# B&R Automation Studio project KeePakST401VersionX
Automation Studio 4.7.5.60 SP; technology packages: Acp10Arnc0 5.8.2, mapp 1.71.0, TextSystem 

## Configuration Config1

CPU X20CP0484, AutomationRuntime C4.72, Build 4.1.2, Vc V4.72.0

### Task classes (Cpu.sw)
```
Cyclic#4 (cycle 100000 us, tolerance 100000 us):
  Program <- Program.prg
  FlexTest <- Actuators.FlexTest.prg
Libraries: AsEPL, runtime, AsBrStr, AsMbTCP, standard, Lib_PBFlx
```

### Hardware
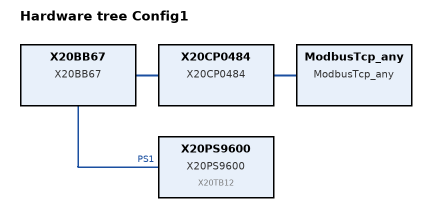
```
ModbusTcp_any : ModbusTcp_any v1.0.6.0  [ETH1 -> X20CP0484.IF2 [Cable Type=PowerlinkCable, Length=10, Version=1.0.0.2]]
  IpAddress = 192.168.0.56
  UnitId = 1
X20BB67 : X20BB67 v1.1.0.0
  Connector IF6:
    CycleTime = 4000
X20CP0484 : X20CP0484 v1.2.1.0  [SL -> X20BB67.SL1]
  Connector IF2:
    ActivateDevice = 1
    Mode = Manual
    InternetAddress = 192.168.0.137
    SubnetMask = 255.255.255.0
    InaNodeNumber = 3
    ActivateModbus = 1
    NumSlaves = -1
    NumAllBlocks = -1
    MemSizeIn = -1
    MemSizeOut = -1
    SlaveDiagnostics = 1
  ConfigurationID = PBFlex_PL_Test1_Config1
  TimerDeviceType = SWIOTIMER
  Cyclic1Duration = 10000
  Cyclic1Tolerance = 10000
  Cyclic2Duration = 20000
  Cyclic2Tolerance = 20000
  Cyclic3Duration = 50000
  Cyclic3Tolerance = 50000
  Cyclic4Duration = 100000
  Cyclic4Tolerance = 100000
  Cyclic5Duration = 200000
  Cyclic5Tolerance = 200000
  Cyclic6Duration = 500000
  Cyclic6Tolerance = 500000
  Cyclic7Duration = 1000000
  Cyclic7Tolerance = 1000000
  Cyclic8Duration = 10000
  Cyclic8Tolerance = 30000000
X20PS9600 : X20PS9600 v1.0.1.0  [PS -> X20BB67.PS1; SS1 -> X20TB12.SS]
X20TB12 : X20TB12 v1.0.0.0
```

### IoMap.iom - X20CP0484/IoMap.iom
```iecst
VAR_CONFIG
	::i_arr_Input_Flex[0] AT %IW."ModbusTcp_any".StateData1;
	::i_arr_Input_Flex[1] AT %IW."ModbusTcp_any".StateData2;
	::i_arr_Output_Flex[0] AT %QW."ModbusTcp_any".CtrWord;
	::b_ModuleStatus AT %IX."ModbusTcp_any".ModuleOk;
END_VAR
```

## Configuration MasterConfiguration_ServoRam

CPU X20CP0484, AutomationRuntime C4.72, Build 4.1.2, Safety 1.10, Vc V4.72.0

### Task classes (Cpu.sw)
```
Cyclic#1 (cycle 4000 us, tolerance 0 us):
  ModeContro <- ModeControl.ModeControl_ST.prg
Cyclic#2 (cycle 8000 us, tolerance 8000 us):
  AdhesiveCo <- Actuators.AdhesiveControl.prg
  FoldPushCo <- Actuators.FoldPushControl.prg
  VacuumCont <- Actuators.VacuumControl.prg [disabled]
  ServoRamHa <- ServoMotion.ServoRamHandler.prg
  ServoFeedH <- ServoMotion.ServoFeedHandler.prg
  ServoHoppe <- ServoMotion.ServoHopperHandler.prg
  MotionHand <- ServoMotion.MotionHandler.prg
  MappCalls <- ServoMotion.MappCalls.prg
Cyclic#3 (cycle 48000 us, tolerance 48000 us):
  SafetySamp <- AsSafetySolution.SafetySample.prg
Cyclic#4 (cycle 100000 us, tolerance 100000 us):
  FlexTest1 <- Actuators.FlexTest.prg
Cyclic#8 (cycle 4000 us, tolerance 30000000 us):
  Recipes <- Recipes.Recipes.prg
  HMIControl <- HMI.HMIControl.prg
  AlarmHandl <- AlarmControl.AlarmHandling.prg
  FlexTest <- Actuators.NordsonComm.NordsonMBComm.prg
  NordsonExt <- Actuators.NordsonComm.NordsonExtendedComm.prg
  PatliteCom <- Stacklight.PatliteComm.prg
  GluePattCt <- Recipes.GluePattCtrl.prg
DataObjects: assl1, Acp10sys
NcDataObjects: acp10etxen <- ServoMotion.acp10etxen.dob, gHopa <- gFeedobj.gHopa.dob, gFeedi <- gFeedobj.gFeedi.dob
VcDataObjects: Visu <- HMI.Visu.dob, Panel <- AsSafetySolution.Panel.dob
Binaries: vccbtn, vcpdvnc, arialbd, vcmgr, vctcal, vcgclass, vcfile, vcctext, vccnum, TCData, vcpkat, udbdef, vcfntttf, arial, vccshape, vcalarm, vccpwd, vcdsloc, Visu01, vccdt, vccscale, vcchspot, vccbmp, vccstr, vcshared, vcrt, vcnet, Visu02, calibri, vcbclass, vcdsint, vcpdsw, vccovl, Visu03, vccddbox, vccpopup, Panel03, Panel02, vcchtml, Panel01, vcxml, vccurl, arsvcreg, TCLang, vcpfgen, vcclbox, Acp10map, acp10cfg, ServoHop, ServoFeed, ServoRam, sysconf, AlarmCfg, RcpCfg, Role, User, ashwd, iomap, arconfig, AlrmHstCfg, TC, asfw, ashwac, vcpdi815, vcptelo, vcpdihd, vcpk, vcpfppc7, vcpdi855, vcpfar00, TopLinMot, BotLinMot, RamCfg
Libraries: operator, runtime, astime, AsIecCon, standard, brsystem, sys_lib, Constants, Vacuum, FoldPush, GluePatt, SetRamPars, GrayToBin, AsBrStr, InvErrTxt, DistCalc, AsSafety, FileIO, AsXml, AsMbTcp, asstring, AsIOAcc, AsBrMath, Lib_PBFlx, AsEPL, DataObj, AsIODiag, Acp10man, Acp10par, NcGlobal, Acp10sdc, Acp10sim, Acp10_MC, MpAxis, MpBase, MpAlarmX, MpCom, MpRecipe, MappCall, Types, AxisFUBs, vcresman, areventlog, powerlnk
```

### Hardware
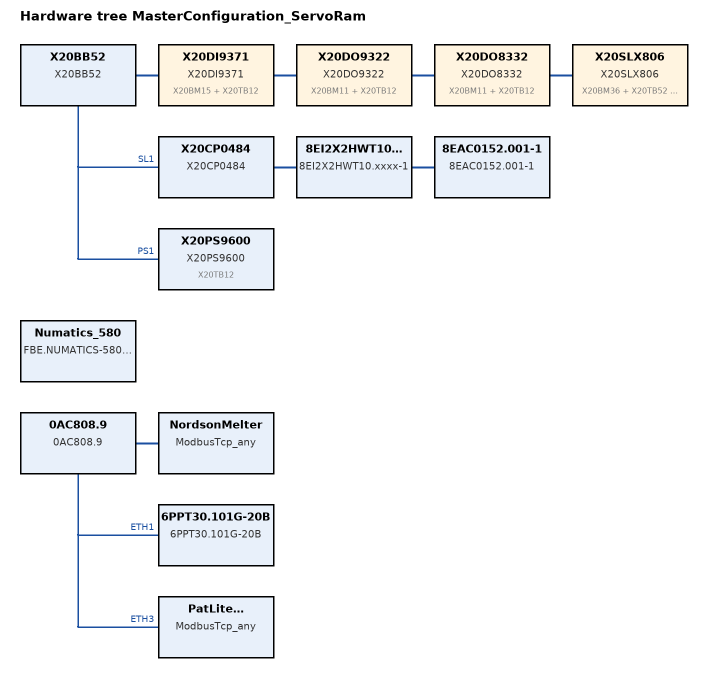
```
0AC808.9 : 0AC808.9 v1.0.0.0  [ETH1 -> 6PPT30.101G-20B.ETH1 [Cable Type=PowerlinkCable, Length=10, Version=1.0.0.2]; ETH2 -> NordsonMelter.ETH1 [Cable Type=PowerlinkCable, Length=10, Version=1.0.0.2]; ETH3 -> PatLite_LightStack.ETH1 [Cable Type=PowerlinkCable, Length=10, Version=1.0.0.2]]
6PPT30.101G-20B : 6PPT30.101G-20B v1.2.0.0  [ETH1 -> 0AC808.9.ETH1 [Cable Type=PowerlinkCable, Length=10, Version=1.0.0.2]; ETH2 -> X20CP0484.IF2 [Cable Type=PowerlinkCable, Length=10, Version=1.0.0.2]]
  Terminal = true
  Startmode = 1
  ShowBootlogoVNC = 1
  Mode = Manual
  InternetAddress = 192.168.0.222
  Subnetmask = 255.255.255.0
  Buttonusage = 1
  ButtonOverride = 1
  ButtonOverrideValue = 2147
  SelectedFavoriteVNC = 192.168.0.100:5900
  Favorites_VNC1 = 192.168.0.100:5900  // Machine Display
  Favorites_VNC2 = 192.168.0.100:5901  // Safety Setup
  PasswordVNC = 2147
  PasswordCIFS = 
  PasswordServiceEncrypt = 1
  PasswordServiceEncrypted = Sr1m/ubkTobKtMGmYG+OdX+pBVPXHNEV0toUjrnwIzvQUaZsN7HbgkMHcdX7NWbHkxunU2zcGZr9hHRCxdVEkcw0t0EkEZxQSM76MpE9s3WvBFtWwy/TiER4jA/5ccmygtG07vdCb9DlCJAeCcJdYe8VLadkZNOaNo2jGOliNnQ=
  VncKeyMappingFile = VC\6PPT30.101G-20B.dis
8EAC0152.001-1 : 8EAC0152.001-1 v2.2.0.1  [SS -> 8EI2X2HWT10.xxxx-1.SS1]
  Ax1PMInterface = Ax1PMEnDat
8EI2X2HWT10.xxxx-1 : 8EI2X2HWT10.xxxx-1 v2.2.0.1  [PLK2 -> X20CP0484.IF3 [Cable Type=PowerlinkCable, Length=10, Version=1.0.0.2]]
  MotionTP = Acp10Arnc0
  EnableDNA = on
  EPL_DNA_Head = 0
  EPL_DNA_HubPort = 1
  EPL_DNA_InPort = 2
  Ax1Interface = Ax1EnDat
  Ax2Interface = Ax2EnDat
  Ax3Interface = Ax3EnDat
NordsonMelter : ModbusTcp_any v1.0.6.0  [ETH1 -> 0AC808.9.ETH2 [Cable Type=PowerlinkCable, Length=10, Version=1.0.0.2]]
  IpAddress = 192.168.0.200
  UnitId = 1
Numatics_580 : FBE.NUMATICS-580-20150428-145500 v1.0 (OrderNumber=Numatics 580)
  Supervision = off
PatLite_LightStack : ModbusTcp_any v1.0.6.0  [ETH1 -> 0AC808.9.ETH3 [Cable Type=PowerlinkCable, Length=10, Version=1.0.0.2]]
  IpAddress = 192.168.0.200
X20BB52 : X20BB52 v1.1.0.0
  Connector IF6:
    CycleTime = 2000
X20BM11 : X20BM11 v1.0.0.1  [X2X1 -> X20BM11d.X2X2]
X20BM11d : X20BM11 v1.0.0.1  [X2X1 -> X20BM15.X2X2]
X20BM15 : X20BM15 v1.0.1.0  [X2X1 -> X20BB52.IF6 (NodeNumber=1)]
X20BM36 : X20BM36 v1.0.0.6  [X2X1 -> X20BM11.X2X2 (NodeNumber=4)]
X20CP0484 : X20CP0484 v1.2.1.0  [SL -> X20BB52.SL1]
  Connector IF2:
    ActivateDevice = 1
    Mode = Manual
    InternetAddress = 192.168.0.100
    SubnetMask = 255.255.255.0
    InaNodeNumber = 0
    Vnc1
    VncVcObjectName1 = Visu
    VncKeyMappingFile1 = VC\PS2-Keyboard.dis
    VncAuthentication1 = 1
    VncPasswordViewOnly1 = 21472147
    VncPasswordViewControl1 = 2147
    VncMaxConnections1 = 4
    VncRefreshRate1 = 100
    Vnc2
    VncVcObjectName2 = Panel
    VncKeyMappingFile2 = VC\PS2-Keyboard1.dis
    VncAuthentication2 = 1
    VncPasswordViewOnly2 = 21472147
    VncPasswordViewControl2 = 2147
    VncPortNumber2 = 5901
    VncRefreshRate2 = 100
    ActivateModbus = 1
    NumSlaves = -1
    NumAllBlocks = -1
    MemSizeIn = -1
    MemSizeOut = -1
  Connector IF3:
    CycleTime = 4000
  ConfigurationID = KeePakVFDCaseErector_C70_10Inch
  UserPartitionSize = 100
  PermanentPvSize = 1024
  RemanentGlobalPvSize = 1024
  TimerDeviceType = EPLX2X
  TimerDevice = X20CP0484.IF3
  TaskClassIdleTime = 4000
  Cyclic1Duration = 4000
  Cyclic1Tolerance = 0
  Cyclic2Duration = 8000
  Cyclic2Tolerance = 8000
  Cyclic3Duration = 48000
  Cyclic3Tolerance = 48000
  Cyclic4Duration = 100000
  Cyclic4Tolerance = 100000
  Cyclic5Duration = 200000
  Cyclic5Tolerance = 200000
  Cyclic6Duration = 500000
  Cyclic6Tolerance = 500000
  Cyclic7Duration = 1000000
  Cyclic7Tolerance = 1000000
  Cyclic8Duration = 4000
  Cyclic8Tolerance = 30000000
  FileDevice1
  FileDeviceName1 = recipes
  FileDevicePath1 = F:\
  EthernetDefaultGateway = 192.168.0.100
  FtpUser1
  FtpUsername1 = jeremy
  FtpUserPassword1 = CB9xa/tRkdxv0VtZFfoX4sbyc2/nOLcpzFFiUfDmX6w=
  FtpUserSalt1 = PVNzvqae
  FTPAccessRight1 = 0
X20DI9371 : X20DI9371 v1.0.2.0  [SS1 -> X20TB12.SS; SL -> X20BM15.SL1]
  Supervision = off
X20DO8332 : X20DO8332 v1.0.2.0  [SS1 -> X20TB12e.SS; SL -> X20BM11.SL1]
  Supervision = off
  PowerSupply01 = on
X20DO9322 : X20DO9322 v1.0.3.0  [SS1 -> X20TB12d.SS; SL -> X20BM11d.SL1]
  Supervision = off
X20PS9600 : X20PS9600 v1.0.1.0  [PS -> X20BB52.PS1; SS1 -> X20TB12f.SS]
X20SLX806 : X20SLX806 v1.10.5.0  [SS1 -> X20TB52.SS; SS2 -> X20TB52a.SS; SL -> X20BM36.SL1]
  Supervision = off
  SafeProject = SafeLOGIC-1
  SafeDesigner = 4.2.6.2
  DigitalOutput01 = viaSafeLOGIC
  DigitalOutput02 = viaSafeLOGIC
  DigitalOutput03 = viaSafeLOGIC
  UnsafeInputUINTs = 4
X20TB12 : X20TB12 v1.0.0.0
X20TB12d : X20TB12 v1.0.0.0
X20TB12e : X20TB12 v1.0.0.0
X20TB12f : X20TB12 v1.0.0.0
X20TB52 : X20TB52 v1.0.0.1
X20TB52a : X20TB52 v1.0.0.1
```

### Cpu.per - X20CP0484/Cpu.per
```iecst
VAR_CONFIG
	ServoFeed_EPD AT %M0; (* *)
	ServoHopper_EPD AT %M40; (* *)
	ServoRam_EPD AT %M80; (* *)
	ServoRamFirstHomeExecuted AT %MX120; (* *)
	ServoFeedFirstHomeExecuted AT %MX121; (* *)
	ServoHopperFirstHomeExecuted AT %MX122; (* *)
	CycleCount AT %MD124; (* *)
	LubeCount AT %MD128; (* *)
END_VAR
```

### IoMap.iom - X20CP0484/IoMap.iom
```iecst
VAR_CONFIG
	Cyclic#1.::gIO.ModuleOKs[4] AT %IX."X20DO8332".ModuleOk;
	Cyclic#1.::gIO.DOs.GlueChannel1 AT %QX."X20DO8332".DigitalOutput01;
	Cyclic#1.::gIO.DOs.GlueChannel2 AT %QX."X20DO8332".DigitalOutput02;
	Cyclic#1.::gIO.DOs.GlueChannel3 AT %QX."X20DO8332".DigitalOutput03;
	Cyclic#1.::gIO.DOs.GlueChannel4 AT %QX."X20DO8332".DigitalOutput04;
	Cyclic#1.::gIO.DOs.ZeroEncoder AT %QX."X20DO8332".DigitalOutput08;
	Cyclic#1.::gIO.DOs.ResetSafety AT %QX."X20SLX806".BOOL101;
	Cyclic#1.::gIO.DIs.SafetyOK AT %IX."X20SLX806".BOOL001;
	Cyclic#1.::gIO.SafetyStatus.CabinetEStopStatus AT %IW."X20SLX806".UINT001;
	Cyclic#1.::gIO.SafetyStatus.SafetyProgramRunning AT %QX."X20SLX806".BOOL102;
	Cyclic#1.::gIO.SafetyStatus.SafetyProgramRunning AT %IX."X20SLX806".BOOL002;
	Cyclic#1.::gIO.ModuleOKs[6] AT %IX."X20SLX806".ModuleOk;
	Cyclic#1.::gIO.ModuleOKs[7] AT %IX."X20SC2212".ModuleOk;
	Cyclic#1.::gIO.SafetyStatus.GuardDoorsOK AT %IX."X20SLX806".BOOL003;
	Cyclic#1.::gIO.SafetyStatus.FrontEStopOK AT %IX."X20SLX806".BOOL004;
	Cyclic#1.::gIO.SafetyStatus.BackEstopOK AT %IX."X20SLX806".BOOL005;
	::gIO.DIs.AdhesivePhotoEye AT %IX."X20DI9371".DigitalInput01;
	::gIO.DIs.DownstreamSensorRaw AT %IX."X20DI9371".DigitalInput04;
	::gIO.DIs.AirPressureOK AT %IX."X20DI9371".DigitalInput03;
	::gIO.DIs.BodyDetect AT %IX."X20DI9371".DigitalInput05;
	::gIO.DIs.AdhesivePhotoEye_2 AT %IX."X20DI9371".DigitalInput02;
	::gIO.ModuleOKs[2] AT %IX."X20DI9371".ModuleOk;
	::gIO.DIs.X_PickRetracted AT %IX."X20DI9371".DigitalInput09;
	::gIO.DIs.X_PickExtended AT %IX."X20DI9371".DigitalInput10;
	::gIO.DIs.X_BlowOff AT %IX."X20DI9371".DigitalInput11;
	::gIO.DIs.BodyHopperLow AT %IX."X20DI9371".DigitalInput06;
	::gIO.DIs.HopperMotor_RUN AT %IX."X20DI9371".DigitalInput07;
	::gIO.DIs.HopperMotor_OFF AT %IX."X20DI9371".DigitalInput08;
	::gIO.DIs.LubricationCounter AT %IX."X20DI9371".DigitalInput12;
	::gIO.DOs.X_PickSolenoid AT %QX."X20DO9322".DigitalOutput03;
	::gIO.DOs.BlowOffOn AT %QX."X20DO9322".DigitalOutput01;
	::gIO.DOs.VacuumOn AT %QX."X20DO9322".DigitalOutput02;
	::gIO.DOs.PushOn AT %QX."X20DO9322".DigitalOutput04;
	::gIO.DOs.RedLightStack AT %QX."X20DO9322".DigitalOutput05;
	::gIO.DOs.GreenLightStack AT %QX."X20DO9322".DigitalOutput06;
	::gIO.DOs.AmberLightStack AT %QX."X20DO9322".DigitalOutput07;
	::gIO.DOs.AirOn AT %QX."X20DO9322".DigitalOutput08;
	Cyclic#1.::gIO.DOs.Pneumatics580ControlWord1 AT %QW."Numatics_580".Out01_I3201Out;
	Cyclic#1.::gIO.ModuleOKs[7] AT %IX."Numatics_580".ModuleOk;
	Cyclic#1.::gIO.DIs.Pneumatics580StatusWord3 AT %IW."Numatics_580".In03_I3403;
	::b_ModuleStatus AT %IX."NordsonMelter".ModuleOk;
END_VAR
```

### Acp10cfg.ncc - X20CP0484/Motion/Acp10cfg.ncc
```
NcConfiguration (Version=5.08.2, NcSwId=Acp10)
  ACP10CF1_typ:
    cnt_nettrc_rec_drive = 1500
    bufsize_trace_upload = 1200
    tc_nc_man_task = Cyclic #1
    glob_pv_as_ncobject = Yes
    ncsys_dl_broadcast = Yes
    ncsys_dl_acp_reset = Yes
    safemc_log_err_to_ax = Yes
    network_init:
      ncsw_init_execute = Yes
      automatic_execute = Yes
      node_nr_warning = Yes
      net_err_before_ncact = Yes
    nettrc:
      enter_parsecrec = Yes
      enter_ncaction = Yes
      save_ring_startidx = No
    cam_prof_download:
      cam_dat_dl_parallel = No
      tc_cam_dl_parallel = Task class for NC Manager task
    plk_if[0]:
      if_name = IF1
      tc_CycDat_PLCopen = Task class for NC Manager task
      mc_broadcast_extdat = No
    plk_if[1]:
      if_name = IF3
      tc_CycDat_PLCopen = Task class for NC Manager task
      mc_broadcast_extdat = No
```

### Acp10map.ncm - X20CP0484/Motion/Acp10map.ncm
```
NcMapping (NcSwId=Acp10, DisabledNodesAreHidden=False)
  NcObject 8EI2X2HWT10.xxxx-1_ncV_AXIS1 (ModuleId=8EI2X2HWT10.xxxx-1, Type=ncV_AXIS, Channel=1, Disabled=TRUE, ModuleDisabled=FALSE)
  NcObject gServoFeed (ModuleId=8EI2X2HWT10.xxxx-1, Type=ncAXIS, Channel=1, AcoposSimulation=Off, InitParameter=gFeedi, Disabled=FALSE, ModuleDisabled=FALSE)
  NcObject 8EI2X2HWT10.xxxx-1_ncV_AXIS2 (ModuleId=8EI2X2HWT10.xxxx-1, Type=ncV_AXIS, Channel=2, Disabled=TRUE, ModuleDisabled=FALSE)
  NcObject gServoRam (ModuleId=8EI2X2HWT10.xxxx-1, Type=ncAXIS, Channel=2, AcoposSimulation=Off, InitParameter=gFeedi, Disabled=FALSE, ModuleDisabled=FALSE)
  NcObject 8EI2X2HWT10.xxxx-1_ncV_AXIS3 (ModuleId=8EI2X2HWT10.xxxx-1, Type=ncV_AXIS, Channel=3, Disabled=TRUE, ModuleDisabled=FALSE)
  NcObject gServoHopper (ModuleId=8EI2X2HWT10.xxxx-1, Type=ncAXIS, Channel=3, AcoposSimulation=Off, InitParameter=gFeedi, AcoposParameter=gHopa, Disabled=FALSE, ModuleDisabled=FALSE)
```

- Safety project (password-protected, skipped)

### AlarmCfg.mpalarmxcore - X20CP0484/mapp/AlarmCfg.mpalarmxcore
```
Element gAlarmXCore (Type=mpalarmxcore)
  mapp.AlarmX.Core:
    Mapping:
      [0]:
        Alarm = Adhesive*
        [0] = Reaction
          Name = AdhesiveAlarm
      [1]:
        Alarm = Vacuum*
        [0] = Reaction
          Name = VacuumAlarm
      [2]:
        Alarm = Air*
        [0] = Reaction
          Name = AirAlarm
      [3]:
        Alarm = Safety*
        [0] = Reaction
          Name = SafetyAlarm
      [4]:
        Alarm = Bliss*
        [0] = Reaction
          Name = BlissPanelAlarm
    BySeverity:
      [0]:
        Severity = 110
        [0] = Reaction
          Name = HighSeverityAlarmActive
      [1]:
        Severity = 1
        [0] = Reaction
          Name = LowSeverityAlarmActive
  mapp.AlarmX.Core.Configuration:
    [0]:
      Name = VacuumPressureLow
      Message = {$AlarmTexts/VacuumPressureLow}
      Code = 1
      Behavior = PersistentAlarm
        ReactionUntilAcknowledged = FALSE
    [1]:
      Name = VacuumOverTemp
      Message = {$AlarmTexts/VacuumOverTemp}
      Code = 1
      Behavior = PersistentAlarm
    [2]:
      Name = AdhesiveUnitNotReady
      Message = {$AlarmTexts/AdhesiveUnitNotReady}
      Code = 2
      Behavior = DiscreteValueMonitoring
        Acknowledge = 0
        ReactionUntilAcknowledged = FALSE
        Monitoring:
          MonitoredPV = ::AdhesiveCo:AdhesiveUnitFaultedAlarmActive
          TriggerValues:
            [0] = TRUE
    [3]:
      Name = AdhesiveUnitFault
      Message = {$AlarmTexts/AdhesiveUnitFault}
      Code = 3
      Behavior = PersistentAlarm
        ReactionUntilAcknowledged = FALSE
    [4]:
      Name = AdhesiveUnitLevelLow
      Message = {$AlarmTexts/AdhesiveUnitLevelLow}
      Code = 4
      Behavior = PersistentAlarm
        ReactionUntilAcknowledged = FALSE
    [5]:
      Name = AdhesiveUseageLow
      Message = {$AlarmTexts/AdhesiveUseageLow}
      Code = 5
      Behavior = PersistentAlarm
        ReactionUntilAcknowledged = FALSE
    [6]:
      Name = AirPressureLow
      Message = {$AlarmTexts/AirPressureLow}
      Code = 6
      Behavior = PersistentAlarm
        ReactionUntilAcknowledged = FALSE
    [7]:
      Name = SafetyNotOK
      Message = {$AlarmTexts/SafetyNotOK}
      Code = 7
      Severity = 110
      Behavior = PersistentAlarm
    [8]:
      Name = SafetyFrontEStop
      Message = {$AlarmTexts/SafetyFrontEStop}
      Code = 7
      Severity = 110
      Behavior = PersistentAlarm
    [9]:
      Name = SafetyBackEStop
      Message = {$AlarmTexts/SafetyBackEStop}
      Code = 7
      Severity = 110
      Behavior = PersistentAlarm
    [10]:
      Name = SafetyGuardDoor
      Message = {$AlarmTexts/SafetyGuardDoor}
      Code = 7
      Severity = 110
      Behavior = PersistentAlarm
        ReactionUntilAcknowledged = FALSE
    [11]:
      Name = VFDAlarm
      Message = {$AlarmTexts/VFDAlarm}
      Code = 8
      Behavior = PersistentAlarm
        ReactionUntilAcknowledged = FALSE
    [12]:
      Name = IOModuleNotOK
      Message = {$AlarmTexts/IOModuleNotOK}
      Code = 9
      Behavior = PersistentAlarm
        ReactionUntilAcknowledged = FALSE
    [13]:
      Name = VFDOverCurrent
      Message = {$AlarmTexts/VFDOverCurrent}
      Behavior = PersistentAlarm
        ReactionUntilAcknowledged = FALSE
    [14]:
      Name = VenturiLow
      Message = {$AlarmTexts/VenturiLow}
      Code = 1
      Behavior = PersistentAlarm
    [15]:
      Name = NordsonComms
      Message = {$AlarmTexts/NordsonComms}
      Behavior = PersistentAlarm
    [16]:
      Name = PatLiteComms
      Message = {$AlarmTexts/PatLiteComms}
      Behavior = PersistentAlarm
    [17]:
      Name = AxisNotHomed
      Message = {$AlarmTexts/AxisNotHomed}
      Behavior = PersistentAlarm
    [18]:
      Name = ATSUnderLimit
      Message = {$AlarmTexts/ATSUnderLimit}
      Behavior = PersistentAlarm
    [19]:
      Name = ATSOverLimit
      Message = {$AlarmTexts/ATSOverLimit}
      Behavior = PersistentAlarm
    [20]:
      Name = AdhesiveNordsonInStandby
      Message = {$AlarmTexts/AdhesiveNordsonInStandby}
      Behavior = PersistentAlarm
    [21]:
      Name = PhotoEyeCheck
      Message = {$AlarmTexts/PhotoEyeCheck}
      Severity = 110
      Behavior = PersistentAlarm
    [22]:
      Name = BodyPanelCheck
      Message = {$AlarmTexts/BodyPanelCheck}
      Severity = 110
      Behavior = DiscreteValueMonitoring
        Monitoring:
          MonitoredPV = ::ModeContro:BodyCheckError
          TriggerValues:
            [0] = TRUE
    [23]:
      Name = HopperLow
      Message = {$AlarmTexts/HopperLow}
      Behavior = DiscreteValueMonitoring
        Acknowledge = 0
        Monitoring:
          MonitoredPV = ::ModeContro:HopperLowAlarm
          InhibitPV = TRUE
          TriggerValues:
            [0] = TRUE
  mapp.AlarmX.Core.Snippets:
    [0]:
      Key = VFDAlarmText
      Value:
        PV = ::gRamCtrlInterface.Status.VFDAlarmText
    [1]:
      Key = IOAlarmText
      Value:
        PV = ::AlarmHandl:IOAlarmText
```

### ServoFeed.mpaxisbasic - X20CP0484/mapp/ServoFeed.mpaxisbasic
```
Element mpServoFeed (Type=mpaxisbasic)
  Alarms = MpAlarmX
    mapp.AlarmX.Core.Configuration:
      [0]:
        Severity = 110
      [1]:
        Severity = 110
      [3]:
        Severity = 110
      [4]:
        Severity = 110
      [6]:
        Severity = 110
      [7]:
        Severity = 110
      [9]:
        Severity = 110
      [11]:
        Severity = 110
      [14]:
        Severity = 110
      [15]:
        Severity = 110
```

### ServoHop.mpaxisbasic - X20CP0484/mapp/ServoHop.mpaxisbasic
```
Element mpServoHopper (Type=mpaxisbasic)
  AxisConfiguration:
    Axis:
      MeasurementUnit = 1
  Alarms = MpAlarmX
    mapp.AlarmX.Core.Configuration:
      [0]:
        Severity = 110
      [1]:
        Severity = 110
      [2]:
        Severity = 110
      [3]:
        Severity = 110
      [4]:
        Severity = 110
      [5]:
        Severity = 110
      [6]:
        Severity = 110
      [7]:
        Severity = 110
      [8]:
        Severity = 110
      [9]:
        Severity = 110
      [10]:
        Severity = 110
      [11]:
        Severity = 110
      [12]:
        Severity = 110
      [13]:
        Severity = 110
      [14]:
        Severity = 110
      [15]:
        Severity = 110
```

### ServoRam.mpaxisbasic - X20CP0484/mapp/ServoRam.mpaxisbasic
```
Element mpServoRam (Type=mpaxisbasic)
  AxisConfiguration:
    Axis:
      MeasurementUnit = 1
  Alarms = MpAlarmX
    mapp.AlarmX.Core.Configuration:
      [0]:
        Severity = 110
      [1]:
        Severity = 110
      [2]:
        Severity = 110
      [3]:
        Severity = 110
      [4]:
        Severity = 110
      [5]:
        Severity = 110
      [6]:
        Severity = 110
      [7]:
        Severity = 110
      [8]:
        Severity = 110
      [9]:
        Severity = 110
      [10]:
        Severity = 110
      [11]:
        Severity = 110
      [12]:
        Severity = 110
      [13]:
        Severity = 110
      [14]:
        Severity = 110
      [15]:
        Severity = 110
```

## Configuration P74_Office

CPU X20CP3585, AutomationRuntime J4.25, Build 4.1.2, Safety 1.10, Vc V4.26.0

### Task classes (Cpu.sw)
```
Cyclic#1 (cycle 2000 us, tolerance 0 us):
  ModeContro <- ModeControl.ModeControl.prg
Cyclic#2 (cycle 10000 us, tolerance 10000 us):
  AdhesiveCo <- Actuators.AdhesiveControl.prg
  FoldPushCo <- Actuators.FoldPushControl.prg
  VacuumCont <- Actuators.VacuumControl.prg
Cyclic#4 (cycle 100000 us, tolerance 100000 us):
  NordsonMBC <- Actuators.NordsonComm.NordsonMBComm.prg [disabled]
  FlexTest <- Actuators.FlexTest.prg
Cyclic#8 (cycle 10000 us, tolerance 30000000 us):
  HMIControl <- HMI.HMIControl.prg
  Recipes <- Recipes.Recipes.prg
  AlarmHandl <- AlarmControl.AlarmHandling.prg
DataObjects: assl1, Acp10sys
NcDataObjects: acp10etxen <- ServoMotion.acp10etxen.dob
VcDataObjects: Visu <- HMI.Visu.dob
Binaries: vccdt, vccbmp, Visu03, vcfile, arial, vctcal, vccpwd, vcrt, vccstr, vcbclass, vccbtn, vcmgr, vcgclass, vcdsint, vcnet, vcpdvnc, vcpfx20, vcshared, arialbd, vccnum, vcpdsw, vccshape, vcctext, Visu01, vcfntttf, vccovl, vcalarm, vcpkat, Visu02, udbdef, calibri, arsvcreg, vcdsloc, vcchspot, TCData, User, sysconf, ashwd, RcpCfg, Role, iomap, asfw, TC, arconfig, RamCfg, AlarmCfg, acp10cfg, Acp10map, vcpk, vcptelo, vcpdi815, vcpdi855, vcpdihd, vcpfppc7
Libraries: powerlnk, vcresman, acp10man, ashw, dataobj, acp10_mc, acp10par
```

### Hardware
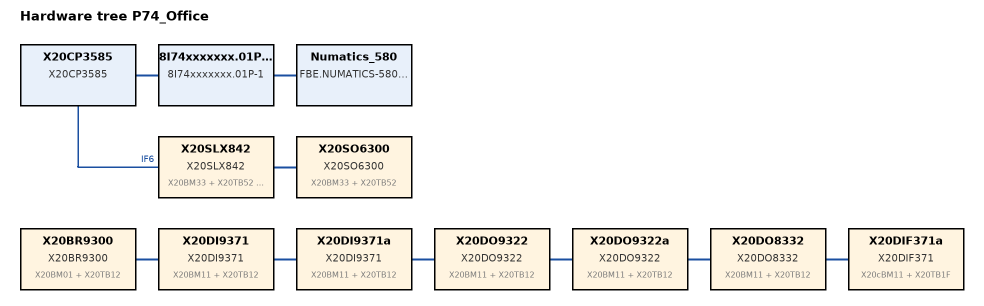
```
8I74xxxxxxx.01P-1 : 8I74xxxxxxx.01P-1 v1.2.0.1  [PLK1 -> X20CP3585.IF3 (NodeNumber=1); PLK2 -> Numatics_580.PLK1 (NodeNumber=1)]
  FunctionModel = Standard
  Supervision = off
  ACC = 2
  DEC = 2
  HSP = 600
  ITH = 20
  BFR = 1
  TFR = 600
  NPR = 5
  UNS = 230
  NCR = 20
  FRS = 600
  NSP = 1750
Numatics_580 : FBE.NUMATICS-580-20150428-145500 v1.0 (Disabled=true, OrderNumber=Numatics 580)  [PLK1 -> 8I74xxxxxxx.01P-1.PLK2 (NodeNumber=2)]
  Supervision = off
X20BM01 : X20BM01 v1.0.1.1 (Disabled=true)
X20BM11 : X20BM11 v1.0.0.1 (Disabled=true)  [X2X1 -> X20BM11f.X2X2]
X20BM11c : X20BM11 v1.0.0.1 (Disabled=true)  [X2X1 -> X20BM01.X2X2]
X20BM11d : X20BM11 v1.0.0.1 (Disabled=true)  [X2X1 -> X20BM11c.X2X2]
X20BM11e : X20BM11 v1.0.0.1 (Disabled=true)  [X2X1 -> X20BM11d.X2X2]
X20BM11f : X20BM11 v1.0.0.1 (Disabled=true)  [X2X1 -> X20BM11e.X2X2]
X20BM33 : X20BM33 v1.0.0.4  [X2X1 -> X20CP3585.IF6]
X20BM33a : X20BM33 v1.0.0.4  [X2X1 -> X20BM33.X2X2]
X20BR9300 : X20BR9300 v1.0.3.0 (Disabled=true)  [SS1 -> X20TB12.SS; SL -> X20BM01.SL1]
  Supervision = off
X20CP3585 : X20CP3585 v1.3.0.0
  Connector IF2:
    ActivateDevice = 1
    EthInterfaceRedundant = 0
    Mode = Manual
    InternetAddress = 192.168.1.100
    SubnetMask = 255.255.255.0
    Vnc1
    VncVcObjectName1 = Visu
    VncKeyMappingFile1 = VC\PS2-Keyboard.dis
    VncAuthentication1 = 1
    VncPasswordViewControl1 = 2147
    VncRefreshRate1 = 100
  Connector IF3:
    EplInterfaceRedundant = 0
    EplEthInterfaceRedundant = 0
  ConfigurationID = KeePakVFDCaseErector_C70_10Inch
  UserPartitionSize = 100
  TimerDeviceType = EPLX2X
  TimerDevice = X20CP3585.IF3
  TaskClassIdleTime = 2000
  Cyclic1Duration = 2000
  Cyclic1Tolerance = 0
  Cyclic2Duration = 10000
  Cyclic2Tolerance = 10000
  Cyclic3Duration = 50000
  Cyclic3Tolerance = 50000
  Cyclic4Duration = 100000
  Cyclic4Tolerance = 100000
  Cyclic5Duration = 200000
  Cyclic5Tolerance = 200000
  Cyclic6Duration = 500000
  Cyclic6Tolerance = 500000
  Cyclic7Duration = 1000000
  Cyclic7Tolerance = 1000000
  Cyclic8Duration = 10000
  Cyclic8Tolerance = 30000000
  FileDevice1
  FileDeviceName1 = recipes
  FileDevicePath1 = F:\
  FtpUser1
  FtpUsername1 = jeremy
  FtpUserPassword1 = CB9xa/tRkdxv0VtZFfoX4sbyc2/nOLcpzFFiUfDmX6w=
  FtpUserSalt1 = PVNzvqae
  FTPAccessRight1 = 0
X20DI9371 : X20DI9371 v1.0.2.0 (Disabled=true)  [SS1 -> X20TB12g.SS; SL -> X20BM11c.SL1]
  Supervision = off
X20DI9371a : X20DI9371 v1.0.2.0 (Disabled=true)  [SS1 -> X20TB12h.SS; SL -> X20BM11d.SL1]
  Supervision = off
X20DIF371a : X20DIF371 v1.0.1.0 (Disabled=true)  [SS1 -> X20TB1F1.SS; SL -> X20cBM11.SL1]
  Supervision = off
X20DO8332 : X20DO8332 v1.0.2.0 (Disabled=true)  [SS1 -> X20TB12e.SS; SL -> X20BM11.SL1]
  Supervision = off
X20DO9322 : X20DO9322 v1.0.3.0 (Disabled=true)  [SS1 -> X20TB12a.SS; SL -> X20BM11e.SL1]
  Supervision = off
X20DO9322a : X20DO9322 v1.0.3.0 (Disabled=true)  [SS1 -> X20TB12b.SS; SL -> X20BM11f.SL1]
  Supervision = off
X20SLX842 : X20SLX842 v1.0.0.0  [SS1 -> X20TB52.SS; SS2 -> X20TB52a.SS; SL -> X20BM33.SL1]
  Supervision = off
  SafeProject = SafeLOGIC-1
  SafeDesigner = 4.2.2.18
X20SO6300 : X20SO6300 v1.10.0.0  [SS1 -> X20TB52b.SS; SL -> X20BM33a.SL1]
  Supervision = off
  DigitalOutput01 = viaSafeLOGIC
  DigitalOutput02 = viaSafeLOGIC
X20TB12 : X20TB12 v1.0.0.0 (Disabled=true)
X20TB12a : X20TB12 v1.0.0.0 (Disabled=true)
X20TB12b : X20TB12 v1.0.0.0 (Disabled=true)
X20TB12e : X20TB12 v1.0.0.0 (Disabled=true)
X20TB12g : X20TB12 v1.0.0.0 (Disabled=true)
X20TB12h : X20TB12 v1.0.0.0 (Disabled=true)
X20TB1F1 : X20TB1F v1.0.0.0 (Disabled=true)
X20TB52 : X20TB52 v1.0.0.1
X20TB52a : X20TB52 v1.0.0.1
X20TB52b : X20TB52 v1.0.0.1
X20cBM11 : X20cBM11 v1.0.0.0 (Disabled=true)  [X2X1 -> X20BM11.X2X2]
```

### IoMap.iom - X20CP3585/IoMap.iom
```iecst
VAR_CONFIG
	Cyclic#1.::gIO.DIs.AdhesivePhotoEye AT %IX."X20DI9371".DigitalInput01;
	Cyclic#1.::gIO.DIs.VacuumTempOK AT %IX."X20DI9371".DigitalInput02;
	Cyclic#1.::gIO.DIs.AirPressureOK AT %IX."X20DI9371".DigitalInput03;
	Cyclic#1.::gIO.DIs.DownstreamSensorRaw AT %IX."X20DI9371".DigitalInput04;
	Cyclic#1.::gIO.DIs.AdhesiveUnitReady AT %IX."X20DI9371".DigitalInput05;
	Cyclic#1.::gIO.DIs.AdhesiveUnitNotFaulted AT %IX."X20DI9371".DigitalInput06;
	Cyclic#1.::gIO.DOs.Pneumatics580ControlWord1 AT %QW."Numatics_580".Out01_I3201Out;
	Cyclic#1.::gIO.DIs.SSI_Parallel.Bits[0] AT %IX."X20DIF371a".DigitalInput01;
	Cyclic#1.::gIO.DIs.SSI_Parallel.Bits[1] AT %IX."X20DIF371a".DigitalInput02;
	Cyclic#1.::gIO.DIs.SSI_Parallel.Bits[2] AT %IX."X20DIF371a".DigitalInput03;
	Cyclic#1.::gIO.DIs.SSI_Parallel.Bits[3] AT %IX."X20DIF371a".DigitalInput04;
	Cyclic#1.::gIO.DIs.SSI_Parallel.Bits[4] AT %IX."X20DIF371a".DigitalInput05;
	Cyclic#1.::gIO.DIs.SSI_Parallel.Bits[5] AT %IX."X20DIF371a".DigitalInput06;
	Cyclic#1.::gIO.DIs.SSI_Parallel.Bits[6] AT %IX."X20DIF371a".DigitalInput07;
	Cyclic#1.::gIO.DIs.SSI_Parallel.Bits[7] AT %IX."X20DIF371a".DigitalInput08;
	Cyclic#1.::gIO.DIs.SSI_Parallel.Bits[8] AT %IX."X20DIF371a".DigitalInput09;
	Cyclic#1.::gIO.DIs.SSI_Parallel.Bits[9] AT %IX."X20DIF371a".DigitalInput10;
	Cyclic#1.::gIO.DIs.SSI_Parallel.Bits[10] AT %IX."X20DIF371a".DigitalInput11;
	Cyclic#1.::gIO.DIs.SSI_Parallel.Bits[11] AT %IX."X20DIF371a".DigitalInput12;
	Cyclic#1.::gIO.DIs.SSI_Parallel.Bits[12] AT %IX."X20DIF371a".DigitalInput13;
	Cyclic#1.::gIO.DIs.SSI_Parallel.Bits[13] AT %IX."X20DIF371a".DigitalInput14;
	Cyclic#1.::gIO.DIs.SSI_Parallel.Bits[14] AT %IX."X20DIF371a".DigitalInput15;
	Cyclic#1.::gIO.ModuleOKs[1] AT %IX."X20BR9300".ModuleOk;
	Cyclic#1.::gIO.ModuleOKs[2] AT %IX."X20DI9371".ModuleOk;
	Cyclic#1.::gIO.ModuleOKs[3] AT %IX."X20DI9371a".ModuleOk;
	Cyclic#1.::gIO.ModuleOKs[4] AT %IX."X20DO9322".ModuleOk;
	Cyclic#1.::gIO.ModuleOKs[5] AT %IX."X20DO9322a".ModuleOk;
	Cyclic#1.::gIO.ModuleOKs[6] AT %IX."X20DO8332".ModuleOk;
	Cyclic#1.::gIO.ModuleOKs[7] AT %IX."X20DIF371a".ModuleOk;
	Cyclic#1.::gIO.ModuleOKs[9] AT %IX."Numatics_580".ModuleOk;
	Cyclic#1.::gIO.DOs.RedLightStack AT %QX."X20DO9322a".DigitalOutput01;
	Cyclic#1.::gIO.DOs.GreenLightStack AT %QX."X20DO9322a".DigitalOutput02;
	Cyclic#1.::gIO.DOs.AmberLightStack AT %QX."X20DO9322a".DigitalOutput03;
	Cyclic#1.::gIO.DOs.AirOn AT %QX."X20DO9322a".DigitalOutput04;
	Cyclic#1.::gIO.DOs.GlueChannel1 AT %QX."X20DO8332".DigitalOutput01;
	Cyclic#1.::gIO.DOs.GlueChannel2 AT %QX."X20DO8332".DigitalOutput02;
	Cyclic#1.::gIO.DOs.GlueChannel3 AT %QX."X20DO8332".DigitalOutput03;
	Cyclic#1.::gIO.DOs.GlueChannel4 AT %QX."X20DO8332".DigitalOutput04;
	Cyclic#1.::gIO.DOs.ResetSafety AT %QX."X20DO9322".DigitalOutput01;
	Cyclic#1.::gIO.DOs.ZeroEncoder AT %QX."X20DO8332".DigitalOutput08;
	Cyclic#1.::gIO.DOs.VacuumOn AT %QX."X20DO9322".DigitalOutput02;
	Cyclic#1.::gIO.DIs.LowAdhesiveUseage AT %IX."X20DI9371a".DigitalInput01;
	Cyclic#1.::gIO.DIs.Pneumatics580StatusWord3 AT %IW."Numatics_580".In03_I3403;
	Cyclic#1.::gIO.DOs.FreeWheelStop AT %QX."X20DO9322".DigitalOutput03;
	::p74Interfa:p74IOInterface.inputs.moduleOK AT %IX."8I74xxxxxxx.01P-1".ModuleOk;
	::p74Interfa:p74IOInterface.inputs.status.readyToSwitchOn AT %IX."8I74xxxxxxx.01P-1".ETAD_Input_Bool_00;
	::p74Interfa:p74IOInterface.inputs.status.switchedOn AT %IX."8I74xxxxxxx.01P-1".ETAD_Input_Bool_01;
	::p74Interfa:p74IOInterface.inputs.status.operationEnabled AT %IX."8I74xxxxxxx.01P-1".ETAD_Input_Bool_02;
	::p74Interfa:p74IOInterface.inputs.status.faultDetection AT %IX."8I74xxxxxxx.01P-1".ETAD_Input_Bool_03;
	::p74Interfa:p74IOInterface.inputs.status.voltageEnabled AT %IX."8I74xxxxxxx.01P-1".ETAD_Input_Bool_04;
	::p74Interfa:p74IOInterface.inputs.status.quickStop AT %IX."8I74xxxxxxx.01P-1".ETAD_Input_Bool_05;
	::p74Interfa:p74IOInterface.inputs.status.switchOnDisabled AT %IX."8I74xxxxxxx.01P-1".ETAD_Input_Bool_06;
	::p74Interfa:p74IOInterface.inputs.status.alarm AT %IX."8I74xxxxxxx.01P-1".ETAD_Input_Bool_07;
	::p74Interfa:p74IOInterface.inputs.spdFeedback AT %IW."8I74xxxxxxx.01P-1".RFRD_Input;
	::p74Interfa:p74IOInterface.inputs.lastFault AT %IW."8I74xxxxxxx.01P-1".LFT_Input;
	::p74Interfa:p74IOInterface.outputs.Commands.switchOn AT %QX."8I74xxxxxxx.01P-1".CMDD_Output_Bool_00;
	::p74Interfa:p74IOInterface.outputs.Commands.enableVoltage AT %QX."8I74xxxxxxx.01P-1".CMDD_Output_Bool_01;
	::p74Interfa:p74IOInterface.outputs.Commands.quickStop AT %QX."8I74xxxxxxx.01P-1".CMDD_Output_Bool_02;
	::p74Interfa:p74IOInterface.outputs.Commands.operationEnable AT %QX."8I74xxxxxxx.01P-1".CMDD_Output_Bool_03;
	::p74Interfa:p74IOInterface.outputs.Commands.faultReset AT %QX."8I74xxxxxxx.01P-1".CMDD_Output_Bool_07;
	::p74Interfa:p74IOInterface.outputs.Commands.stopCommand AT %QX."8I74xxxxxxx.01P-1".CMDD_Output_Bool_08;
	::p74Interfa:p74IOInterface.outputs.Commands.revDirection AT %QX."8I74xxxxxxx.01P-1".CMDD_Output_Bool_11;
	::p74Interfa:p74IOInterface.outputs.spdReference AT %QW."8I74xxxxxxx.01P-1".LFRD_Output;
	::p74Interfa:p74IOInterface.inputs.STO AT %IW."8I74xxxxxxx.01P-1".STOS_Input;
	::gIO.DIs.SafetyOK AT %IX."X20SLX842".BOOL001;
	::gIO.DOs.ResetSafety AT %QX."X20SLX842".BOOL101;
	::gIO.SafetyStatus.SafetyProgramRunning AT %IX."X20SLX842".BOOL002;
END_VAR
```

### Acp10cfg.ncc - X20CP3585/Motion/Acp10cfg.ncc
```
NcConfiguration (Version=3.14.0, NcSwId=Acp10)
  ACP10CF1_typ:
    cnt_nettrc_rec_drive = 150
    bufsize_trace_upload = 1200
    tc_nc_man_task = Cyclic #1
    glob_pv_as_ncobject = Yes
    ncsys_dl_broadcast = Yes
    ncsys_dl_acp_reset = Yes
    safemc_log_err_to_ax = Yes
    network_init:
      ncsw_init_execute = Yes
      automatic_execute = No
      node_nr_warning = Yes
      net_err_before_ncact = Yes
    nettrc:
      enter_parsecrec = Yes
      enter_ncaction = Yes
      save_ring_startidx = No
    cam_prof_download:
      cam_dat_dl_parallel = No
      tc_cam_dl_parallel = Task class for NC Manager task
    sdc_if[0]:
      if_name = SDC_IF1
      mc_broadcast_size = 800
      mc_broadcast_extdat = No
```

### AlarmCfg.mpalarmxcore - X20CP3585/mapp/AlarmCfg.mpalarmxcore
```
Element gAlarmXCore (Type=mpalarmxcore)
  mapp.AlarmX.Core:
    Mapping:
      [0]:
        Alarm = Adhesive*
        [0] = Reaction
          Name = AdhesiveAlarm
      [1]:
        Alarm = Vacuum*
        [0] = Reaction
          Name = VacuumAlarm
      [2]:
        Alarm = Air*
        [0] = Reaction
          Name = AirAlarm
      [3]:
        Alarm = Safety*
        [0] = Reaction
          Name = SafetyAlarm
  mapp.AlarmX.Core.Configuration:
    [0]:
      Name = VacuumPressureLow
      Message = {$AlarmTexts/VacuumPressureLow}
      Code = 1
      Behavior = PersistentAlarm
        ReactionUntilAcknowledged = FALSE
    [1]:
      Name = VacuumOverTemp
      Message = {$AlarmTexts/VacuumOverTemp}
      Code = 1
      Behavior = PersistentAlarm
    [2]:
      Name = AdhesiveUnitNotReady
      Message = {$AlarmTexts/AdhesiveUnitNotReady}
      Code = 2
      Behavior = PersistentAlarm
        ReactionUntilAcknowledged = FALSE
    [3]:
      Name = AdhesiveUnitFault
      Message = {$AlarmTexts/AdhesiveUnitFault}
      Code = 3
      Behavior = PersistentAlarm
        ReactionUntilAcknowledged = FALSE
    [4]:
      Name = AdhesiveUnitLevelLow
      Message = {$AlarmTexts/AdhesiveUnitLevelLow}
      Code = 4
      Behavior = PersistentAlarm
        ReactionUntilAcknowledged = FALSE
    [5]:
      Name = AdhesiveUseageLow
      Message = {$AlarmTexts/AdhesiveUseageLow}
      Code = 5
      Behavior = PersistentAlarm
        ReactionUntilAcknowledged = FALSE
    [6]:
      Name = AirPressureLow
      Message = {$AlarmTexts/AirPressureLow}
      Code = 6
      Behavior = PersistentAlarm
        ReactionUntilAcknowledged = FALSE
    [7]:
      Name = SafetyNotOK
      Message = {$AlarmTexts/SafetyNotOK}
      Code = 7
      Behavior = PersistentAlarm
        ReactionUntilAcknowledged = FALSE
    [8]:
      Name = VFDAlarm
      Message = {$AlarmTexts/VFDAlarm}
      Code = 8
      Behavior = PersistentAlarm
        ReactionUntilAcknowledged = FALSE
    [9]:
      Name = IOModuleNotOK
      Message = {$AlarmTexts/IOModuleNotOK}
      Code = 9
      Behavior = PersistentAlarm
        ReactionUntilAcknowledged = FALSE
    [10]:
      Name = VFDOverCurrent
      Message = {$AlarmTexts/VFDOverCurrent}
      Behavior = PersistentAlarm
        ReactionUntilAcknowledged = FALSE
  mapp.AlarmX.Core.Snippets:
    [0]:
      Key = VFDAlarmText
      Value:
        PV = ::gRamCtrlInterface.Status.VFDAlarmText
    [1]:
      Key = IOAlarmText
      Value:
        PV = ::AlarmHandl:IOAlarmText
```

### RamCfg.mpaxisbasic - X20CP3585/mapp/RamCfg.mpaxisbasic
```
Element mpRamAxis (Type=mpaxisbasic)
  AxisConfiguration = AxisWithConfiguration
    Axis:
      MovementLimits:
        VelocityPositive = 120
        VelocityNegative = 120
        Acceleration = 1500
        Deceleration = 1500
        PositionErrorStopLimit = 5.0
    Drive:
      Gearbox:
        Input = 60
      Controller:
        Position:
          ProportionalGain = 20
          PredictionTime = 0.002
          TotalDelayTime = 0.002
        Speed:
          ProportionalGain = 0.05
        LoopFilters:
          [0]
          [1]
          [2]
  Alarms = MpAlarmX
```

## Configuration Simulation

CPU PC_any, AutomationRuntime F4.26, Build 4.1.2, Vc V4.26.1

### Task classes (Cpu.sw)
```
Cyclic#1 (cycle 2000 us, tolerance 0 us):
  Simulation <- Simulation.Simulation.prg
  ModeContro <- ModeControl.ModeControl.prg
Cyclic#2 (cycle 10000 us, tolerance 10000 us):
  AdhesiveCo <- Actuators.AdhesiveControl.prg
  FolderCont <- Actuators.FoldPushControl.prg
  VacuumCont <- Actuators.VacuumControl.prg
Cyclic#4 (cycle 1000000 us, tolerance 10000000 us):
  EncoderDec <- EncoderDecoding.prg [disabled]
  FlexTest <- Actuators.FlexTest.prg
Cyclic#8 (cycle 8000 us, tolerance 30000000 us):
  HMIControl <- HMI.HMIControl.prg
  AlarmHandl <- AlarmControl.AlarmHandling.prg
  Recipes <- Recipes.Recipes.prg
  NordsonMBC <- Actuators.NordsonComm.NordsonMBComm.prg
DataObjects: Acp10sys
NcDataObjects: acp10etxen <- ServoMotion.acp10etxen.dob, gLinAxisi, gLinAxisa
VcDataObjects: Visu <- HMI.Visu.dob
Binaries: vccdt, vccbmp, Visu03, vcfile, arial, vctcal, vccpwd, vcrt, arsvcreg, vccstr, vcbclass, vccbtn, vcgclass, vcdsint, vcnet, vcmgr, vcshared, arialbd, vccnum, vcpdvnc, vcpdsw, vcpfar00, vcctext, Visu01, vcfntttf, vccovl, vccshape, vcalarm, vcpkat, Visu02, udbdef, calibri, vcdsloc, vcchspot, TCData, vccddbox, vccscale, vccpopup, TopLinMot, BotLinMot, AlrmHstCfg, User, sysconf, ashwd, RcpCfg, Role, iomap, asfw, TC, arconfig, RamCfg, AlarmCfg, Acp10map, acp10cfg, Config, vccalarm, vccbar, vccurl, vcchtml, vccslider, vcctrend, vccline, vcxml
Libraries: powerlnk, vcresman, dataobj, areventlog
```

### Hardware
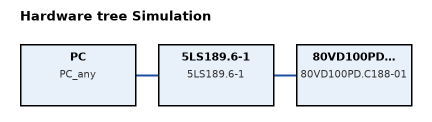
```
5LS189.6-1 : 5LS189.6-1 v1.3.0.0  [SL -> PC.SL1]
  Connector IF2:
    EplEthInterfaceRedundant = 0
80VD100PD.C188-01 : 80VD100PD.C188-01 v2.0.1.0  [PLK1 -> 5LS189.6-1.IF2 (NodeNumber=2)]
  Simulate = standard
PC : PC_any v1.1.0.0 (OrderNumber=PC)
  Connector IF3:
    Vnc1
    VncVcObjectName1 = Visu
    VncKeyMappingFile1 = VC\PS2-Keyboard.dis
    VncAuthentication1 = 1
    VncPasswordViewOnly1 = 21472147
    VncPasswordViewControl1 = 2147
    VncRefreshRate1 = 100
  ConfigurationID = KeePakVFDCaseErector_Config1
  PermanentPvSize = 4096
  SystemTick = 2000
  Cyclic1Duration = 2000
  Cyclic1Tolerance = 0
  Cyclic2Duration = 10000
  Cyclic2Tolerance = 10000
  Cyclic3Duration = 500000
  Cyclic3Tolerance = 10000000
  Cyclic4Duration = 1000000
  Cyclic4Tolerance = 10000000
  Cyclic5Duration = 2000000
  Cyclic5Tolerance = 10000000
  Cyclic6Duration = 3000000
  Cyclic6Tolerance = 12000000
  Cyclic7Duration = 4000000
  Cyclic7Tolerance = 12000000
  Cyclic8Duration = 8000
  Cyclic8Tolerance = 30000000
  FileDevice1
  FileDeviceName1 = recipes
  FileDevicePath1 = C:\Temp\recipe
```

### Cpu.per - PC/Cpu.per
```iecst
VAR_CONFIG
	gEndlessPosBot AT %M0; (*Bottom folder endless position*)
	gEndlessPosTop AT %M40; (*Top folder endless position*)
END_VAR
```

### Acp10cfg.ncc - PC/Motion/Acp10cfg.ncc
```
NcConfiguration (Version=3.18.2, NcSwId=Acp10)
  ACP10CF1_typ:
    cnt_nettrc_rec_drive = 1500
    bufsize_trace_upload = 1200
    tc_nc_man_task = Cyclic #1
    glob_pv_as_ncobject = Yes
    ncsys_dl_broadcast = Yes
    ncsys_dl_acp_reset = Yes
    safemc_log_err_to_ax = Yes
    network_init:
      ncsw_init_execute = Yes
      automatic_execute = No
      node_nr_warning = Yes
      net_err_before_ncact = Yes
    nettrc:
      enter_parsecrec = Yes
      enter_ncaction = Yes
      save_ring_startidx = Yes
    cam_prof_download:
      cam_dat_dl_parallel = No
      tc_cam_dl_parallel = Task class for NC Manager task
    plk_if[0]:
      if_name = SL1.IF2
      tc_CycDat_PLCopen = Task class for NC Manager task
      mc_broadcast_extdat = No
```

### Acp10map.ncm - PC/Motion/Acp10map.ncm
```
NcMapping (NcSwId=Acp10, DisabledNodesAreHidden=False)
  NcObject gTopLinAxis (ModuleId=80VD100PD.C188-01, Type=ncAXIS, Channel=1, AcoposSimulation=Standard, InitParameter=gTopLinAx1, AcoposParameter=gTopLinAxi, Disabled=FALSE, ModuleDisabled=FALSE)
  NcObject gBotLinAxis (ModuleId=80VD100PD.C188-01, Type=ncAXIS, Channel=2, AcoposSimulation=Standard, InitParameter=gBotLinAx1, AcoposParameter=gBotLinAxi, Disabled=FALSE, ModuleDisabled=FALSE)
  NcObject 80VD100PD.C188-01_ncV_AXIS1 (ModuleId=80VD100PD.C188-01, Type=ncV_AXIS, Channel=1, Disabled=TRUE, ModuleDisabled=FALSE)
  NcObject 80VD100PD.C188-01_ncV_AXIS2 (ModuleId=80VD100PD.C188-01, Type=ncV_AXIS, Channel=2, Disabled=TRUE, ModuleDisabled=FALSE)
```

### AlarmCfg.mpalarmxcore - PC/mapp/AlarmCfg.mpalarmxcore
```
Element gAlarmXCore (Type=mpalarmxcore)
  mapp.AlarmX.Core:
    Mapping:
      [0]:
        Alarm = Adhesive*
        [0] = Reaction
          Name = AdhesiveAlarm
      [1]:
        Alarm = Vacuum*
        [0] = Reaction
          Name = VacuumAlarm
      [2]:
        Alarm = Air*
        [0] = Reaction
          Name = AirAlarm
      [3]:
        Alarm = Safety*
        [0] = Reaction
          Name = SafetyAlarm
      [4]:
        Alarm = Bliss*
        [0] = Reaction
          Name = BlissPanelAlarm
  mapp.AlarmX.Core.Configuration:
    [0]:
      Name = VacuumPressureLow
      Message = {$AlarmTexts/VacuumPressureLow}
      Code = 1
      Behavior = PersistentAlarm
        ReactionUntilAcknowledged = FALSE
    [1]:
      Name = VacuumOverTemp
      Message = {$AlarmTexts/VacuumOverTemp}
      Code = 1
      Behavior = PersistentAlarm
    [2]:
      Name = AdhesiveUnitNotReady
      Message = {$AlarmTexts/AdhesiveUnitNotReady}
      Code = 2
      Behavior = PersistentAlarm
        ReactionUntilAcknowledged = FALSE
    [3]:
      Name = AdhesiveUnitFault
      Message = {$AlarmTexts/AdhesiveUnitFault}
      Code = 3
      Behavior = PersistentAlarm
        ReactionUntilAcknowledged = FALSE
    [4]:
      Name = AdhesiveUnitLevelLow
      Message = {$AlarmTexts/AdhesiveUnitLevelLow}
      Code = 4
      Behavior = PersistentAlarm
        ReactionUntilAcknowledged = FALSE
    [5]:
      Name = AdhesiveUseageLow
      Message = {$AlarmTexts/AdhesiveUseageLow}
      Code = 5
      Behavior = PersistentAlarm
        ReactionUntilAcknowledged = FALSE
    [6]:
      Name = AirPressureLow
      Message = {$AlarmTexts/AirPressureLow}
      Code = 6
      Behavior = PersistentAlarm
        ReactionUntilAcknowledged = FALSE
    [7]:
      Name = SafetyNotOK
      Message = {$AlarmTexts/SafetyNotOK}
      Code = 7
      Behavior = PersistentAlarm
    [8]:
      Name = SafetyFrontEStop
      Message = {$AlarmTexts/SafetyFrontEStop}
      Code = 7
      Behavior = PersistentAlarm
    [9]:
      Name = SafetyBackEStop
      Message = {$AlarmTexts/SafetyBackEStop}
      Code = 7
      Behavior = PersistentAlarm
    [10]:
      Name = SafetyGuardDoor
      Message = {$AlarmTexts/SafetyGuardDoor}
      Code = 7
      Behavior = PersistentAlarm
        ReactionUntilAcknowledged = FALSE
    [11]:
      Name = VFDAlarm
      Message = {$AlarmTexts/VFDAlarm}
      Code = 8
      Behavior = PersistentAlarm
        ReactionUntilAcknowledged = FALSE
    [12]:
      Name = IOModuleNotOK
      Message = {$AlarmTexts/IOModuleNotOK}
      Code = 9
      Behavior = PersistentAlarm
        ReactionUntilAcknowledged = FALSE
    [13]:
      Name = VFDOverCurrent
      Message = {$AlarmTexts/VFDOverCurrent}
      Behavior = PersistentAlarm
        ReactionUntilAcknowledged = FALSE
    [14]:
      Name = BlissSidePanelCheck
      Message = {$AlarmTexts/BlissSidePanelCheck}
      Behavior = PersistentAlarm
    [15]:
      Name = BlissBodyCheck
      Message = {$AlarmTexts/BlissBodyCheck}
      Behavior = PersistentAlarm
    [16]:
      Name = VenturiLow
      Message = {$AlarmTexts/VenturiLow}
      Code = 1
      Behavior = PersistentAlarm
    [17]:
      Name = NordsonComms
      Message = {$AlarmTexts/NordsonComms}
      Behavior = PersistentAlarm
    [18]:
      Name = PatLiteComms
      Message = {$AlarmTexts/PatLiteComms}
      Behavior = PersistentAlarm
    [19]:
      Name = AxisNotHomed
      Message = {$AlarmTexts/AxisNotHomed}
      Behavior = PersistentAlarm
    [20]:
      Name = ATSUnderLimit
      Message = {$AlarmTexts/ATSUnderLimit}
      Behavior = PersistentAlarm
    [21]:
      Name = ATSOverLimit
      Message = {$AlarmTexts/ATSOverLimit}
      Behavior = PersistentAlarm
  mapp.AlarmX.Core.Snippets:
    [0]:
      Key = VFDAlarmText
      Value:
        PV = ::gRamCtrlInterface.Status.VFDAlarmText
    [1]:
      Key = IOAlarmText
      Value:
        PV = ::AlarmHandl:IOAlarmText
```

### AlrmHstCfg.mpalarmxhistory - PC/mapp/AlrmHstCfg.mpalarmxhistory
```
Element gAlarmXHistory (Type=mpalarmxhistory)
  mapp.AlarmX.History:
    Memory:
      MemorySize = 60
```

### BotLinMot.mpaxisbasic - PC/mapp/BotLinMot.mpaxisbasic
```
Element gBotAxisBasic (Type=mpaxisbasic)
  Alarms = MpAlarmX
```

### RamCfg.mpaxisbasic - PC/mapp/RamCfg.mpaxisbasic
```
Element mpRamAxis (Type=mpaxisbasic)
  AxisConfiguration = AxisWithConfiguration
    Axis:
      MovementLimits:
        VelocityPositive = 150
        VelocityNegative = 150
        Acceleration = 1500
        Deceleration = 1500
    Drive:
      Controller:
        Position:
          ProportionalGain = 20
        Speed:
          ProportionalGain = 0.05
        LoopFilters:
          [0]
          [1]
          [2]
  Alarms = MpAlarmX
```

### TopLinMot.mpaxisbasic - PC/mapp/TopLinMot.mpaxisbasic
```
Element gTopAxisBasic (Type=mpaxisbasic)
  Alarms = MpAlarmX
```

## Logical view

Binary libraries used (declarations not repeated): operator, runtime, astime, AsIecCon, standard, brsystem, sys_lib, AsBrStr, AsSafety, FileIO, AsXml, AsMbTCP, asstring, AsIOAcc, AsBrMath, AsEPL, DataObj, AsIODiag, Acp10man 5.08.2, Acp10par 5.08.2, NcGlobal 5.08.2, Acp10sdc 5.08.2, Acp10sim 5.08.2, Acp10_MC 5.08.2, MpAxis 1.71.0, MpBase 5.08.0, MpAlarmX 1.71.0, MpCom 1.71.0, MpRecipe 1.71.0

### Global.var - Global variables
```iecst
VAR
	TON_RamDelay : TON; (*Timer for the Ram to delay forward motion*)
	StopFeed : BOOL;
END_VAR
VAR RETAIN
	ServoRam_EPD : MC_ENDLESS_POSITION;
END_VAR
VAR
	ServoRamTrigger : BOOL;
END_VAR
VAR RETAIN
	ServoRamFirstHomeExecuted : BOOL;
END_VAR
VAR
	ServoRamClear : BOOL;
	ServoRamBusy : BOOL;
	ServoRamAutoHome : BOOL;
END_VAR
VAR RETAIN
	ServoHopper_EPD : MC_ENDLESS_POSITION;
	ServoHopperFirstHomeExecuted : BOOL;
	ServoFeed_EPD : MC_ENDLESS_POSITION;
	ServoFeedFirstHomeExecuted : BOOL;
END_VAR
VAR
	RamDelay : TIME;
	PhotoEyeSeen : BOOL;
	Melter : DUT_NDSN_Flex;
	LubricationOK : BOOL;
END_VAR
VAR RETAIN
	LubeCount : UDINT;
END_VAR
VAR
	InfeedBoxPresent : BOOL;
	HopperLowTime : TIME := T#7s;
	HoperLowStop : BOOL;
	gVacCtrlInterface : VacCtrlInterface_typ;
	gUserLevel : USINT;
	gTopLinAxis_1 : ACP10AXIS_typ;
	gTopLinAxis : ACP10AXIS_typ;
	gSoftwareReset : BOOL;
	gServoRamInterface : Axis_Interface_typ;
	gServoRam : ACP10AXIS_typ;
	gServoHopperInterface : Axis_Interface_typ;
	gServoHopper : ACP10AXIS_typ;
	gServoFeedInterface : Axis_Interface_typ;
	gServoFeed : ACP10AXIS_typ;
	gSafetyNotOKAlarmActive : BOOL;
END_VAR
VAR RETAIN
	gRecipeInterface : {REDUND_UNREPLICABLE} RecipeCtrlInterface_typ := (0);
END_VAR
VAR
	gRamCtrlInterface : RamControlInterface_typ;
	gRamAtStopPosition : BOOL;
	gPusherOn : BOOL;
	gPassword : ARRAY[0..2] OF STRING[80] := ['','1111','2147'];
	gOnDelayCompensation : REAL;
	gOffDelayCompensation : REAL;
	gNumAlarms : UDINT;
	gNumActiveAlarms : UDINT;
	gModeControlInterface : ModeCtrlInterface_typ;
	gLowSeverityAlarmActive : BOOL;
	gIsSimulated : BOOL;
	gIO : IO_typ;
	gHomingParameters : Home_Parameters_typ;
	gHMI : HMIControl_typ;
	gHighSeverityAlarmActive : BOOL;
	gFoldPushCtrlInterface : FoldPushCtrlInterface_typ := (Parameters:=(LinMotBotFolder:=(Parameter:=(MpBasicParameters:=(Home:=(Mode:=mpAXIS_HOME_MODE_RESTORE_POS,Position:=0,StartVelocity:=25,HomingVelocity:=5,Acceleration:=500,StartDirection:=mpAXIS_HOME_DIR_NEGATIVE,TorqueLimit:=0.5,BlockDetectionPositionError:=4,PositionErrorStopLimit:=10),Jog:=(Velocity:=2)))),LinMotTopFolder:=(Parameter:=(MpBasicParameters:=(Home:=(Mode:=mpAXIS_HOME_MODE_RESTORE_POS,Position:=0,StartVelocity:=25,HomingVelocity:=5,Acceleration:=500,StartDirection:=mpAXIS_HOME_DIR_NEGATIVE,TorqueLimit:=0.5,BlockDetectionPositionError:=4,PositionErrorStopLimit:=10),Jog:=(Velocity:=2))))));
END_VAR
VAR RETAIN
	gEndlessPosTop : MC_ENDLESS_POSITION;
	gEndlessPosBot : MC_ENDLESS_POSITION;
END_VAR
VAR
	gDownstreamBlocked : BOOL;
	gCurrentLimitHit : BOOL;
	gChangePage : USINT;
	gBotLinAxis_1 : ACP10AXIS_typ;
	gBotLinAxis : ACP10AXIS_typ;
	gAutoTune : BOOL;
	gAlarmSystemActive : BOOL;
	gAlarmActive : BOOL;
	gAirPressureAlarmActive : BOOL;
	gAdhesiveCtrlInterface : AdhesiveCtrlInterface_typ;
	gActivePage : USINT;
	FeedServoBusy : BOOL;
	FeedPositionCapture : LREAL;
	FeedPosFinal : LREAL;
	FeedInCycle : BOOL;
	DistanceAfterLatch : REAL;
END_VAR
VAR RETAIN
	CycleCount : UDINT;
END_VAR
VAR
	b_ModuleStatus : BOOL;
END_VAR
```

### Package Logical/Libraries - Global libraries

### Library Logical/Libraries/Constants (IEC)

#### Constants.var - Exported constants
```iecst
VAR CONSTANT
	COUNTS_PER_ENCODER_REV : UINT := 23040;
	DEFAULT_RECIPE_NAME : STRING[255] := 'settings.xml';
	HIDE : USINT := 1;
	LOCK : USINT := 2;
	MAX_NUM_GLUE_CHANNELS : USINT := 4;
	MAX_NUM_GLUE_CHANNELS_M1 : USINT := MAX_NUM_GLUE_CHANNELS-1;
	MAX_NUM_ONOFF_PATTERNS : USINT := 4;
	MAX_NUM_ONOFF_PATTERNS_M1 : USINT := MAX_NUM_ONOFF_PATTERNS-1;
	NOTOK : USINT := 0;
	OK : USINT := 1;
	PPM_TO_DEG_PER_S : REAL := 6.0;
	UNHIDE : USINT := 0;
	UNLOCK : USINT := 0;
	ALARM_INACTIVE : USINT := 0;
	ALARM_ACTIVE : USINT := 1;
	PAGE_ALARM : USINT := 100;
	PUMPS_OFF : USINT := 16#0;
	PUMPS_ON : USINT := 16#2;
	MELTER_OFF : USINT := 16#0;
	MELTER_ON : USINT := 16#1;
	STANDBY_ON : USINT := 16#40; (*bit 6 on*)
	WRITE_COMMAND : USINT := 16#6;
	READ_COMMAND : USINT := 16#3;
	TEMP_UNIT_IDX : USINT := 110;
	TEMP_UNIT_START_CHANNEL : USINT := 0;
	IDX_SET_TEMP : USINT := 115;
	CHANNEL_SET_TEMP_START : USINT := 1;
	IDX_MELTER_STATUS : USINT := 10;
	IDX_ATS_ALARMS : USINT := 229;
	IDX_ACT_TEMP : USINT := 120;
	CHANNEL_ACT_TEMP_START : USINT := 1;
	IDX_ADHESIVE_HOUR : USINT := 225;
	CHANNEL_ADHESIVE_HOUR : USINT := 0;
	MAX_NUM_TEMP_CHANNELS : USINT := 5;
	MAX_NUM_TEMP_CHANNELS_M1 : USINT := MAX_NUM_TEMP_CHANNELS-1;
	MACHINE_TYPE_BLISS : USINT := 3;
	MACHINE_TYPE_CLASSICPAK : USINT := 1;
	MACHINE_TYPE_TRAY : USINT := 2;
	NUM_NORDSON_TEMP_ZONES : USINT := 6;
	NUM_NORDSON_TEMP_ZONES_M1 : USINT := NUM_NORDSON_TEMP_ZONES-1;
	TYPE1_RECIPE_NAME : STRING[80] := 'settings1.xml';
	TYPE2_RECIPE_NAME : STRING[80] := 'settings2.xml';
END_VAR
```

#### AlarmNames.var
```iecst
VAR CONSTANT
	ALARM_ADHESIVE_FAULT : STRING[255] := 'AdhesiveUnitFault';
	ALARM_ADHESIVE_LOW : STRING[255] := 'AdhesiveUnitLevelLow';
	ALARM_ADHESIVE_NOT_READY : STRING[255] := 'AdhesiveUnitNotReady';
	ALARM_VACUUM_OVER_TEMP : STRING[255] := 'VacuumOverTemp';
	ALARM_VACUUM_PRESSURE_LOW : STRING[255] := 'VacuumPressureLow';
	ALARM_AIR_PRESSURE_LOW : STRING[255] := 'AirPressureLow';
	ALARM_SAFETY_NOTOK : STRING[255] := 'SafetyNotOK';
	ALARM_VFD : STRING[255] := 'VFDAlarm';
	ALARM_IO_MODULE_NOT_OK : STRING[255] := 'IOModuleNotOK';
	ALARM_ADHESIVE_USEAGE_LOW : STRING[255] := 'AdhesiveUseageLow';
	ALARM_VFD_OVER_CURRENT : STRING[255] := 'VFDOverCurrent';
	ALARM_TEST_ALARM2 : STRING[255] := 'TestAlarm2';
	ALARM_TEST_ALARM : STRING[255] := 'TestAlarm';
	ALARM_VENTURI_LOW : STRING[255] := 'VenturiLow';
	ALARM_NORDSON_COMMS : STRING[255] := 'NordsonComms';
	ALARM_SAFETY_FRONT_ESTOP : STRING[255] := 'SafetyFrontEStop';
	ALARM_SAFETY_REAR_ESTOP : STRING[255] := 'SafetyBackEStop';
	ALARM_SAFETY_GUARD_DOOR : STRING[255] := 'SafetyGuardDoor';
	ALARM_PATLITE_COMMS : STRING[255] := 'PatLiteComms';
	ALARM_NOT_HOMED : STRING[255] := 'AxisNotHomed';
	ALARM_ATS_UNDERLIMIT : STRING[255] := 'ATSUnderLimit';
	ALARM_ATS_OVERLIMIT : STRING[255] := 'ATSOverLimit';
	ALARM_NORDSON_STANDBY : STRING[255] := 'AdhesiveNordsonInStandby';
	ALARM_PHOTOEYE_CHECK : STRING[255] := 'PhotoEyeCheck';
	ALARM_BODY_CHECK : STRING[255] := 'BodyPanelCheck';
END_VAR
```

### Library Logical/Libraries/Vacuum (IEC)

#### Vacuum.fun - Exported functions and function blocks
```iecst
FUNCTION VenturiControl : BOOL (*Venturi Control*) (*$GROUP=User,$CAT=User,$GROUPICON=User.png,$CATICON=User.png*)
	VAR_INPUT
		Enable : BOOL;
		EncoderPosition : REAL;
		OnPos : REAL;
		OffPos : REAL;
	END_VAR
END_FUNCTION
```

#### VenturiControl.st
```iecst
(* Venturi Control *)
FUNCTION VenturiControl

	IF(Enable = FALSE) THEN
		VenturiControl := FALSE;
	ELSE

		//if on pos equal to off position, do not turn on vacuum
		IF(OnPos = OffPos) THEN
			RETURN;
		END_IF

		IF((EncoderPosition >= OnPos) AND (EncoderPosition <= OffPos)) THEN
			VenturiControl := TRUE;
		END_IF
	END_IF

END_FUNCTION
```

### Library Logical/Libraries/FoldPush (IEC)

#### FoldPush.fun - Exported functions and function blocks
```iecst
FUNCTION FoldPushControl : BOOL (*Fold Push Control*) (*$GROUP=User,$CAT=User,$GROUPICON=User.png,$CATICON=User.png*)
	VAR_INPUT
		EncoderPosition : REAL;
		OnPos : REAL;
		OffPos : REAL;
	END_VAR
END_FUNCTION
```

#### FoldPushControl.st
```iecst
(* Fold Push Control *)
FUNCTION FoldPushControl

	FoldPushControl := FALSE;

	//if on pos equal to off position, do not turn on pushers/folders
	IF(OnPos = OffPos) THEN
		RETURN;
	END_IF

	IF((EncoderPosition >= OnPos) AND (EncoderPosition <= OffPos)) THEN
		FoldPushControl := TRUE;
	END_IF

END_FUNCTION
```

### Library Logical/Libraries/GluePatt (IEC)
Depends on: Types

#### Types.typ - Exported data types
```iecst
TYPE
	Switches : 	STRUCT
		FirstOnPosition : ARRAY[0..MAX_NUM_BEADS_M1]OF REAL;
		LastOnPosition : ARRAY[0..MAX_NUM_BEADS_M1]OF REAL;
	END_STRUCT;
END_TYPE
```

#### Constants.var - Exported constants
```iecst
VAR CONSTANT
	MAX_NUM_BEADS : USINT := 64;
	MAX_NUM_BEADS_M1 : USINT := MAX_NUM_BEADS-1;
END_VAR
```

#### GluePatt.fun - Exported functions and function blocks
```iecst
FUNCTION GluePatternControl : BOOL (*Turns glue channel on off at assigned positions*) (*$GROUP=User,$CAT=User,$GROUPICON=User.png,$CATICON=User.png*)
	VAR_INPUT
		ChannelPattern : AdhesivePattern_typ;
		PositionInCycle : REAL;
		StitchPercentage : REAL;
		BeadLengths : ARRAY[0..MAX_NUM_ONOFF_PATTERNS_M1] OF REAL;
		OnDelayCompensation : REAL;
		OffDelayCompensation : REAL;
		Switches : REFERENCE TO ARRAY[0..MAX_NUM_ONOFF_PATTERNS_M1] OF Switches;
		ChannelModulationCtrl : INT;
	END_VAR
	VAR
		i : USINT;
		j : INT;
		NumOfBeads : ARRAY[0..MAX_NUM_ONOFF_PATTERNS_M1] OF INT;
		GlueLength : ARRAY[0..MAX_NUM_ONOFF_PATTERNS_M1] OF REAL;
		GapLength : ARRAY[0..MAX_NUM_ONOFF_PATTERNS_M1] OF REAL;
		EndCapLength : ARRAY[0..MAX_NUM_ONOFF_PATTERNS_M1] OF REAL;
	END_VAR
END_FUNCTION

FUNCTION SetPatternSDPs : BOOL (*Sets adhesive pattern SDPs based on machine parameters and conditions*) (*$GROUP=User,$CAT=User,$GROUPICON=User.png,$CATICON=User.png*)
	VAR_INPUT
		NumGlueChannels : USINT;
		FieldColormaps : REFERENCE TO ColorMapDatapoints_typ;
		FieldSDPs : REFERENCE TO StatusDatapoints_typ;
	END_VAR
	VAR
		j : INT;
		i : USINT;
	END_VAR
END_FUNCTION
```

#### GluePatternControl.st
```iecst
(* Determines when a glue channel should be turned on/off for a given glue pattern *)
FUNCTION GluePatternControl

	GluePatternControl := FALSE; //set output false. If the cycle position falls within one of our patterns, we'll turn it on

	//  Creating glue stitching patterns
	FOR i := 0 TO MAX_NUM_ONOFF_PATTERNS_M1 DO
		IF ChannelPattern.GlueOnDistance[i] > 0 THEN

			IF BeadLengths[i] = 0 THEN
				BeadLengths[i] := 0.25;
			END_IF;

			IF ChannelModulationCtrl = 0 THEN
				StitchPercentage := 1;
			END_IF;

			// Calculating a pattern's parameters
			GlueLength[i] := ChannelPattern.GlueOnDistance[i] * StitchPercentage;
			IF BeadLengths[i] > GlueLength[i] THEN
				BeadLengths[i] := GlueLength[i];
			ELSIF TRUNC(GlueLength[i] / BeadLengths[i]) > MAX_NUM_BEADS_M1 THEN
				BeadLengths[i] := GlueLength[i] / MAX_NUM_BEADS;
			END_IF;
			NumOfBeads[i] := TRUNC(GlueLength[i] / BeadLengths[i]);
			GapLength[i] := (ChannelPattern.GlueOnDistance[i] - GlueLength[i]) / NumOfBeads[i];
			EndCapLength[i] := GlueLength[i] - (BeadLengths[i] * NumOfBeads[i]);

			// Assigning the on and off locations for a stitch pattern
			FOR j := 0 TO NumOfBeads[i] - 1 DO
				Switches[i].FirstOnPosition[j] := ChannelPattern.DelayDistance[i] + (j * (BeadLengths[i] + GapLength[i]));
				Switches[i].LastOnPosition[j] := ChannelPattern.DelayDistance[i] + (j * (BeadLengths[i] + GapLength[i]) + BeadLengths[i]);
			END_FOR;

			// Adding endcap on and off locations if a pattern has one
			IF EndCapLength[i] <> 0 THEN
				Switches[i].FirstOnPosition[NumOfBeads[i]] := ChannelPattern.DelayDistance[i] + (NumOfBeads[i] * (BeadLengths[i] + GapLength[i]));
				Switches[i].LastOnPosition[NumOfBeads[i]] := ChannelPattern.DelayDistance[i] + (NumOfBeads[i] * (BeadLengths[i] + GapLength[i]) + EndCapLength[i]);

				FOR j := NumOfBeads[i] + 1 TO MAX_NUM_BEADS_M1 DO
					Switches[i].FirstOnPosition[j] := Switches[i].LastOnPosition[j] := 0;
				END_FOR;
			ELSIF NumOfBeads[i] < MAX_NUM_BEADS THEN
				FOR j := NumOfBeads[i] TO MAX_NUM_BEADS_M1 DO
					Switches[i].FirstOnPosition[j] := Switches[i].LastOnPosition[j] := 0;
				END_FOR;
			END_IF;
		ELSE
			FOR j := 0 TO MAX_NUM_BEADS_M1 DO
				Switches[i].FirstOnPosition[j] := Switches[i].LastOnPosition[j] := 0;
			END_FOR;
		END_IF;
	END_FOR;

	//loop over each gluing location's switch points
	//turn on the channel IF we are within a glueing window (adjusted for on/off delays)
	FOR i:=0 TO MAX_NUM_ONOFF_PATTERNS_M1 DO
		FOR j := 0 TO NumOfBeads[i] DO
			IF (ChannelPattern.GlueOnDistance[i] <= 0) THEN
				RETURN;
			ELSIF (((Switches[i].FirstOnPosition[j] - OnDelayCompensation) <= PositionInCycle) AND (PositionInCycle < (Switches[i].LastOnPosition[j] - OffDelayCompensation))) THEN
				GluePatternControl := TRUE;
				RETURN;
			END_IF;
		END_FOR;
	END_FOR;

END_FUNCTION
```

#### SetPatternSDPs.st
```iecst
(* Sets adhesive pattern SDPs based on machine parameters and conditions *)
FUNCTION SetPatternSDPs

	FOR i:=0 TO MAX_NUM_GLUE_CHANNELS_M1 DO
		FOR j:=0 TO MAX_NUM_ONOFF_PATTERNS_M1 DO

			//find a SDP that indicates the edit popup is open (bit 12). Set the colordata point of that field to 1
			IF(FieldSDPs.AdhesiveChannelSDPs[i].Delay[j].12 = 1) THEN
				FieldColormaps.AdhesiveChannelsColormaps[i].Delay[j] := 1;
			ELSE
				FieldColormaps.AdhesiveChannelsColormaps[i].Delay[j] := 0;
			END_IF

			IF(FieldSDPs.AdhesiveChannelSDPs[i].Glue[j].12 = 1) THEN
				FieldColormaps.AdhesiveChannelsColormaps[i].Glue[j] := 1;
			ELSE
				FieldColormaps.AdhesiveChannelsColormaps[i].Glue[j] := 0;
			END_IF

			//hide rows if there are not enough active channels
			IF(NumGlueChannels >= (i+1)) THEN
				FieldSDPs.AdhesiveChannelSDPs[i].RowLabel := UNHIDE + UNLOCK;
				FieldSDPs.AdhesiveChannelSDPs[i].Delay[j].0 := 0; //unhide and unlock
				FieldSDPs.AdhesiveChannelSDPs[i].Delay[j].1 := 0;
				FieldSDPs.AdhesiveChannelSDPs[i].Glue[j].0 := 0;
				FieldSDPs.AdhesiveChannelSDPs[i].Glue[j].1 := 0;
			ELSE
				FieldSDPs.AdhesiveChannelSDPs[i].RowLabel := HIDE + LOCK;
				FieldSDPs.AdhesiveChannelSDPs[i].Delay[j].0 := 1; //hide and lock
				FieldSDPs.AdhesiveChannelSDPs[i].Delay[j].1 := 1;
				FieldSDPs.AdhesiveChannelSDPs[i].Glue[j].0 := 1;
				FieldSDPs.AdhesiveChannelSDPs[i].Glue[j].1 := 1;
			END_IF

		END_FOR;
	END_FOR;

		SetPatternSDPs := 1;

END_FUNCTION
```

### Library Logical/Libraries/SetRamPars (IEC)
Depends on: Types, MpAxis

#### SetRamPars.fun - Exported functions and function blocks
```iecst
FUNCTION SetRamPars : USINT (*Transfer ram movement parameters from the control interface to the motion control block*) (*$GROUP=User,$CAT=User,$GROUPICON=User.png,$CATICON=User.png*)
	VAR_INPUT
		InterfacePars : RamCtrlInterface_Parameters_typ;
		MotionPars : REFERENCE TO MpAxisBasicParType;
	END_VAR
END_FUNCTION

FUNCTION ComputeMoveDistance : REAL (*Computes how far the ram should go in order to reach the stop position*) (*$GROUP=User,$CAT=User,$GROUPICON=User.png,$CATICON=User.png*)
	VAR_INPUT
		TargetPos : REAL;
		CurrentPos : REAL;
	END_VAR
END_FUNCTION

FUNCTION ComputeDistanceMoved : REAL (*Compute how far encoder has moved*) (*$GROUP=User,$CAT=User,$GROUPICON=User.png,$CATICON=User.png*)
	VAR_INPUT
		CurentPos : REAL;
		OldPos : REAL;
	END_VAR
END_FUNCTION
```

#### SetRamPars.st
```iecst
(* Transfer ram movement parameters from the control interface to the motion control block *)
FUNCTION SetRamPars

	MotionPars.Acceleration := InterfacePars.Acceleration;
	MotionPars.Deceleration := InterfacePars.Acceleration;
	MotionPars.Position := InterfacePars.Position;
	MotionPars.Direction := mpAXIS_DIR_POSITIVE;

	MotionPars.Jog.Acceleration := InterfacePars.Acceleration;
	MotionPars.Jog.Deceleration := InterfacePars.Acceleration;
	MotionPars.Jog.Velocity := InterfacePars.JogSpeed;

	SetRamPars := 1;

END_FUNCTION
```

#### ComputeMoveDistance.st
```iecst
(* Computes how far the ram should go in order to reach the stop position *)
FUNCTION ComputeMoveDistance

	IF((TargetPos -  CurrentPos) > 0) THEN
		ComputeMoveDistance := TargetPos -  CurrentPos;
	ELSE
		ComputeMoveDistance := 360.0 + TargetPos -  CurrentPos;
	END_IF

END_FUNCTION
```

#### ComputeDistanceMoved.st
```iecst
(* Compute how far encoder has moved *)
FUNCTION ComputeDistanceMoved

	IF((CurentPos -  OldPos) >= 0) THEN
		ComputeDistanceMoved := CurentPos -  OldPos;
	ELSE
		ComputeDistanceMoved := 360.0 + CurentPos -  OldPos;
	END_IF

END_FUNCTION
```

### Library Logical/Libraries/GrayToBin (ANSIC)

#### GrayToBin.fun - Exported functions and function blocks
```iecst
FUNCTION grayToBinary : UDINT (*Convert gray code to binary*) (*$GROUP=User,$CAT=User,$GROUPICON=User.png,$CATICON=User.png*)
	VAR_INPUT
		bits : ARRAY[0..15] OF BOOL;
	END_VAR
END_FUNCTION

FUNCTION grayCodeBitPacker : UDINT (*packs gray code bits into a single variable*) (*$GROUP=User,$CAT=User,$GROUPICON=User.png,$CATICON=User.png*)
	VAR_INPUT
		bits : ARRAY[0..15] OF BOOL;
	END_VAR
END_FUNCTION
```

#### GrayToBinary.c
```c
#include <bur/plctypes.h>
#include "grayToBin.h"

#ifdef __cplusplus
	extern "C"
	{
#endif

#ifdef __cplusplus
	};
#endif

/* Convert gray code to binary */
unsigned long grayToBinary(plcbit bits[16])
{

	unsigned long num;
	//	unsigned int mask;
	//	for (mask = num >> 1; mask != 0; mask = mask >> 1)
	//	{
	//		num = num ^ mask;
	//	}
	//	return num;

	num = grayCodeBitPacker(bits);

	num = num ^ (num >> 16);
	num = num ^ (num >> 8);
	num = num ^ (num >> 4);
	num = num ^ (num >> 2);
	num = num ^ (num >> 1);
	return num;
}
```

#### grayCodeBitPacker.c
```c
#include <bur/plctypes.h>
#ifdef __cplusplus
	extern "C"
	{
#endif
	#include "GrayToBin.h"
#ifdef __cplusplus
	};
#endif

/* packs gray code bits into a single variable */
unsigned long grayCodeBitPacker(plcbit bits[16])
{
	UDINT BitPackedGrayCode = 0;
	unsigned short i;

	for (i = 0; i < 16; i++)
	{
		BitPackedGrayCode = BitPackedGrayCode | (bits[i] << i);
	}

	return BitPackedGrayCode;
}
```

### Library Logical/Libraries/InvErrTxt (IEC, version 1.00.1) - This library takes in the error number from the AcoposInverter I/O datapoint mapping screen and returns a text description
Depends on: asstring

#### InvErrTxt.typ - Exported data types
```iecst
(********************************************************************
 * COPYRIGHT --
 ********************************************************************
 * Library: InvErrTxt
 * File: InvErrTxt.typ
 * Author: scoccimaroj
 * Created: November 09, 2010
 ********************************************************************
 * Data types of library InvErrTxt
 ********************************************************************)

TYPE
	ACPInverterFaultText_typ : 	STRUCT  (*structure definition for the input types to the FUB*)
		FaultNumber : INT; (*variable definition for the input passed into the FUB that identifies which element in the error text array is to be displayed*)
		FaultDescription : STRING[64]; (*variable definition for the input passed into the FUB that displays the string text of the fault error text of the drive fault*)
	END_STRUCT;
	EACPInverterType_enum :
		( (*enumeration definition for the selection of the inverter drive types available for use with this FUB*)
		EACPInverter_S44 := 0, (*enum member definition for the S44 inverter*)
		EACPInverter_X64 := 1, (*enum member definition for the X64 inverter*)
		EACPInverter_P84 := 2, (*enum member definition for the P84 inverter*)
		EACPInverter_P74 := 3 (*enum member definition for the P74 inverter*)
		);
	InvErrTxtStatus_enum :
		( (*enumeration definition for the output of the FUB to display the current status of the FUB*)
		INACTIVE := 0, (*enum member definition for when the FUB is inactive, occurs prior to the error text initialization status*)
		INITIALIZING_ERROR_TEXT := 1, (*enum member definition for when the FUB is intitializing the error text, only runs once at start up*)
		IDLE := 2, (*enum member definition for when the FUB is idle while waiting for a fault to occur*)
		BUSY := 3, (*enum member definition for when the FUB is busy processing the fault number to get the fault description*)
		ERROR := 4 (*enum member definition for when the FUB is in error  ***not connected****)
		);
END_TYPE
```

#### InvErrTxt.fun - Exported functions and function blocks
```iecst
(********************************************************************
 * COPYRIGHT --
 ********************************************************************
 * Library: InvErrTxt
 * File: InvErrTxt.fun
 * Author: scoccimaroj
 * Created: November 09, 2010
 ********************************************************************
 * Functions and function blocks of library InvErrTxt
 ********************************************************************)

FUNCTION_BLOCK InverterFaultText
	VAR_INPUT
		Execute : BOOL; (*When TRUE, the error code is read and a matching error text is displayed. Should be tied to a drive faulted boolean*)
		DriveType : EACPInverterType_enum; (*The type of acopos inverter being used.*)
		FaultText : UDINT; (*The address of the string to write the error message to. String must be atleast 64 characters long.*)
		FaultNumber : REFERENCE TO INT; (*Fault number to decode. Given as an address*)
	END_VAR
	VAR_OUTPUT
		Status : InvErrTxtStatus_enum; (*Status of the function block. Read from an enum defined in the typ file of this library*)
		LastFault : INT; (*Output variable for displaying the last fault that was detected on the drive*)
	END_VAR
	VAR
		isInitialized : BOOL; (*Internal Variable.*)
		S44FaultTable : ARRAY[0..35] OF ACPInverterFaultText_typ; (*Internal Variable. Holds S44 fault info.*)
		X64FaultTable : ARRAY[0..31] OF ACPInverterFaultText_typ; (*Internal Variable. Holds X64 fault info.*)
		P84FaultTable : ARRAY[0..74] OF ACPInverterFaultText_typ; (*Internal Variable. Holds P84 fault info.*)
		P74FaultTable : ARRAY[0..66] OF ACPInverterFaultText_typ; (*Internal Variable. Holds P74 fault info.*)
		PreviousFault : INT; (*Internal Variable. Holds the previous fault passed in.*)
		i : USINT; (*Internal Variable.*)
	END_VAR
END_FUNCTION_BLOCK
```
